TYPE DUT_TIMESET :
STRUCT

	sTempTimeYYMMDD: STRING;
	sTempTimeHO: STRING;
	sTempTimeMI: STRING;
	sTempTimeSe: STRING;
END_STRUCT
END_TYPE

(* stored: Version 1.1.0.1, ProductVersion 3.1.4024.9
   DUT DUT_TIMESET: Id {ebb617ca-6cce-47fb-918c-be2b713fecce} *)
